{attribute 'GeneratedUsingTerminal: EL3201-0030-0022'}
{attribute addProperty BoxType "EL3201-0030-0022"}
{attribute addProperty Id "StatusAT %I*Status_F2CE6D917ValueAT %I*INT2"}
{attribute addProperty CRC "1245267073"}
{attribute addProperty Size "9"}
TYPE RTD_4A394481 :
STRUCT
	{attribute addProperty Name "Status"}
	Status AT %I* : Status_F2CE6D91;
	{attribute addProperty Name "Value"}
	Value AT %I* : INT;
END_STRUCT
END_TYPE

(* stored: Version 1.2.0.0, ProductVersion 3.1.4024.9
   DUT RTD_4A394481: Id {c2f12daf-54cd-47f6-8c85-47e38b52d7b9} *)
